FUNCTION_BLOCK DEV_HMI (* Simple Device Front Panel *)
  (* Standard: 61499 Feasibility Demo ITA; Description: Simple Device Front Panel *)
  (* Version 0.1, 2001-06-02, JHC, Rockwell Automation, Replaced IN,OUT_WSTRING to IN,OUT_ANY *)
  (* Version 0.0, 2001-01-08, JHC, Rockwell Automation *)
  (* Compiler header: package fb.rt.ita; import fb.rt.hmi.*; *)
  (* Compiler Java IBM VisualAge 3.0 *)
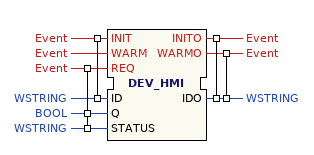
  EVENT_INPUT
    INIT WITH ID; (* Interface Initialization *)
    WARM; (* Warm Restart,User-provided ID *)
    REQ WITH Q, STATUS; (* Manager Status Change *)
  END_EVENT
  EVENT_OUTPUT
    INITO WITH IDO; (* Initialization Confirm *)
    WARMO WITH IDO; (* WARM Restart confirmation *)
  END_EVENT
  VAR_INPUT
    ID : WSTRING := "localhost:61499"; (* Management Socket ID *)
    Q : BOOL; (* Manager QO *)
    STATUS : WSTRING; (* Manager Status *)
  END_VAR
  VAR_OUTPUT
    IDO : WSTRING; (* Initial or user-entered ID *)
  END_VAR
  FBS
    IDIN : IN_ANY;
    QOUT : OUT_BOOL;
    STATOUT : OUT_ANY;
  END_FBS
  EVENT_CONNECTIONS
    INIT TO IDIN.INIT;
    IDIN.INITO TO QOUT.INIT;
    QOUT.INITO TO STATOUT.INIT;
    STATOUT.INITO TO INITO;
    WARM TO IDIN.REQ;
    IDIN.IND TO WARMO;
    REQ TO QOUT.REQ;
    QOUT.CNF TO STATOUT.REQ;
  END_CONNECTIONS
  DATA_CONNECTIONS
    1 TO IDIN.QI;
    1 TO QOUT.QI;
    1 TO STATOUT.QI;
    24 TO IDIN.W;
    16 TO STATOUT.W;
    ID TO IDIN.IVAL;
    Q TO QOUT.IN;
    COLOR#red TO QOUT.C0;
    COLOR#green TO QOUT.C1;
    STATUS TO STATOUT.IN;
    IDIN.OUT TO IDO;
  END_CONNECTIONS
END_FUNCTION_BLOCK
